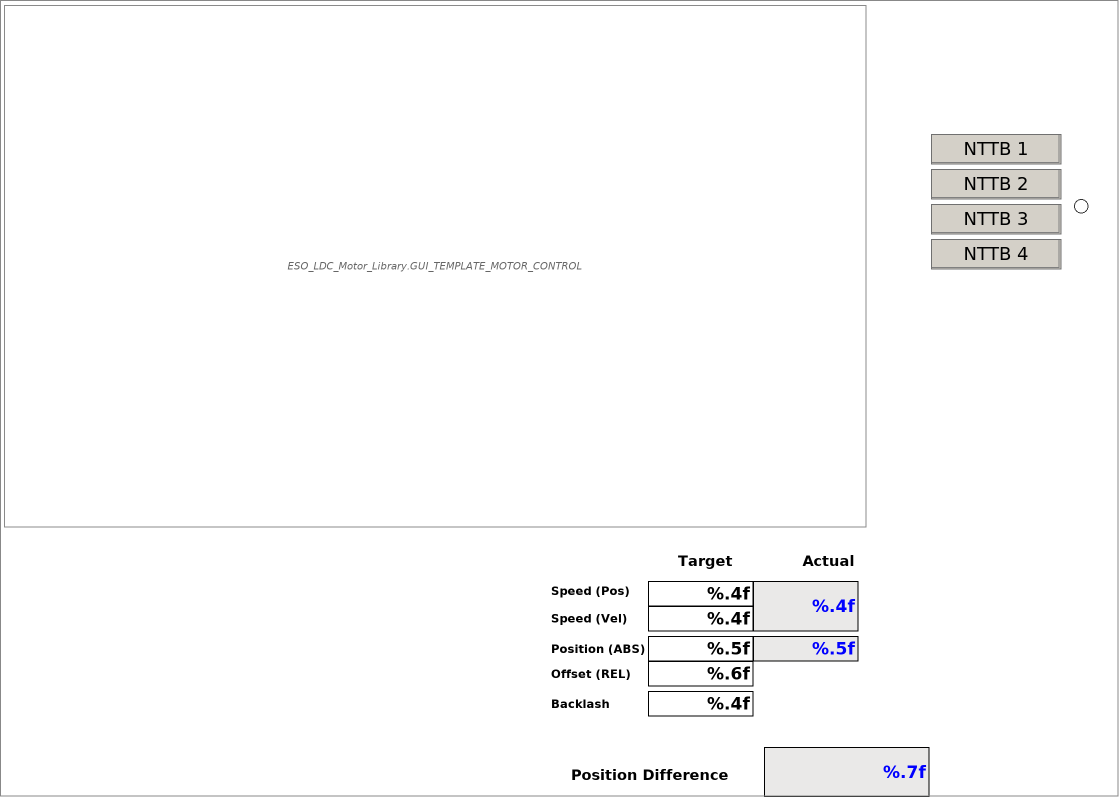
VISUALIZATION GUI_NOTT_TILT_B_CTRL  // 1119x797
    Frame (4,5 862x522)
        shows ESO_LDC_Motor_Library.GUI_TEMPLATE_MOTOR_CONTROL(m_Instance := MAIN.nott_ics.TipTilt.ptrTiltActuatorsB[MAIN.nott_ics.TipTilt.guiTiltActuatorsBIndex]^)
    Rectangle (548,581 95x20), "Speed (Pos)"
    Rectangle (753,636 105x25), "%.5f", text variable: MAIN.nott_ics.Delay_Lines.ptrDelayLines[MAIN.nott_ics.Delay_Lines.guiShutterIndex]^.stat.lrPosActual, input disabled if: false
    Rectangle (675,551 190x20), "Target Actual"
    Rectangle (548,639 95x20), "Position (ABS)"
    Rectangle (753,581 105x50), "%.4f", text variable: MAIN.nott_ics.Delay_Lines.ptrDelayLines[MAIN.nott_ics.Delay_Lines.guiShutterIndex]^.stat.lrVelActual, input disabled if: false
    Rectangle (648,606 105x25), "%.4f", text variable: MAIN.nott_ics.Delay_Lines.ptrDelayLines[MAIN.nott_ics.Delay_Lines.guiShutterIndex]^.ctrl.lrVelocity
        OnMouseDown: write the text variable via Default
    Rectangle (548,694 95x20), "Backlash"
    Rectangle (648,691 105x25), "%.4f", text variable: MAIN.nott_ics.Delay_Lines.ptrDelayLines[MAIN.nott_ics.Delay_Lines.guiShutterIndex]^.cfg.lrBacklash
        OnMouseDown: write the text variable via Default
    Rectangle (548,606 95x25), "Speed (Vel)"
    Rectangle (648,636 105x25), "%.5f", tooltip "Absolute position used by "MOVE ABS"", text variable: MAIN.nott_ics.Delay_Lines.ptrDelayLines[MAIN.nott_ics.Delay_Lines.guiShutterIndex]^.ctrl.lrPosition
        OnMouseDown: write the text variable via Default
    Rectangle (648,581 105x25), "%.4f", text variable: MAIN.nott_ics.Delay_Lines.ptrDelayLines[MAIN.nott_ics.Delay_Lines.guiShutterIndex]^.cfg.lrDefaultVelocity
        OnMouseDown: write the text variable via Default
    Rectangle (548,664 95x20), "Offset (REL)"
    Rectangle (648,661 105x25), "%.6f", tooltip "Relative offset used by "MOVE REL"", text variable: MAIN.nott_ics.Delay_Lines.ptrDelayLines[MAIN.nott_ics.Delay_Lines.guiShutterIndex]^.ctrl.lrOffset
        OnMouseDown: write the text variable via Default
    Rectangle (764,747 165x50), "%.7f", text variable: MAIN.nott_ics.Delay_Lines.ptrDelayLines[MAIN.nott_ics.Delay_Lines.guiShutterIndex]^.stat.lrPosError, input disabled if: false
    Rectangle (568,765 190x20), "Position Difference"
    RadioButton (1072,136 47x140), variable: MAIN.nott_ics.TipTilt.guiTiltActuatorsBIndex-1
        Areas[0]: Text=Radiobutton
        Areas[1]: Text=Radiobutton
    Button (931,134 130x30), "NTTB 1"
        OnMouseClick: execute { MAIN.nott_ics.TipTilt.guiTiltActuatorsBIndex := 1; }
    Button (931,169 130x30), "NTTB 2"
        OnMouseClick: execute { MAIN.nott_ics.TipTilt.guiTiltActuatorsBIndex := 2; }
    Button (931,204 130x30), "NTTB 3"
        OnMouseClick: execute { MAIN.nott_ics.TipTilt.guiTiltActuatorsBIndex := 3; }
    Button (931,239 130x30), "NTTB 4"
        OnMouseClick: execute { MAIN.nott_ics.TipTilt.guiTiltActuatorsBIndex := 4; }
END_VISUALIZATION

// ---- VISUs/Templates/MOTOR_CONTROL.TcVIS
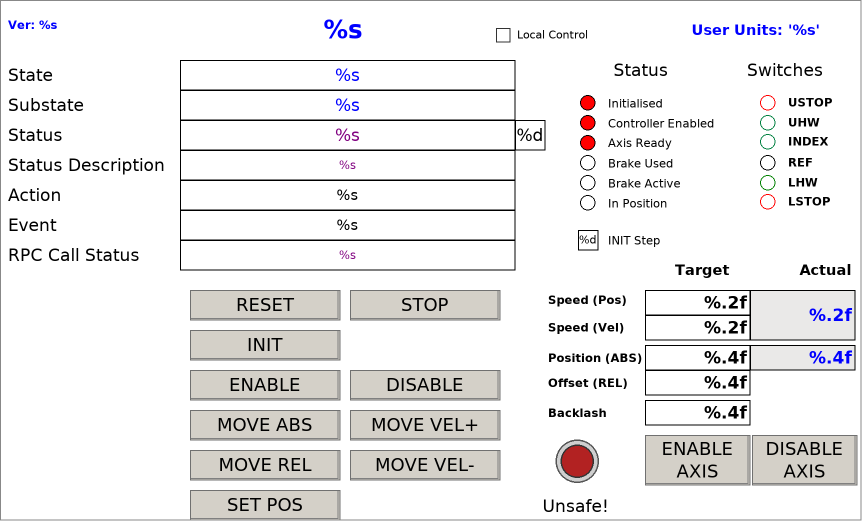
VISUALIZATION MOTOR_CONTROL  // 862x521
VAR_IN_OUT
	m_Instance:	FB_MOTOR;
END_VAR
    Rectangle (180,60 335x30), "%s", text variable: m_Instance.stat.sState
    Rectangle (180,90 335x30), "%s", text variable: m_Instance.stat.sSubstate
    Button (190,290 150x30), "RESET", input disabled if: NOT m_Instance.stat.bLocal OR NOT m_Instance.in_bSafe
        OnMouseDown: execute {
            m_Instance.ctrl.bLocalCmd := TRUE;
            m_Instance.ctrl.nCommand := E_MOTOR_COMMAND.RESET;
            m_Instance.ctrl.bExecute := TRUE;
        }
    Button (190,330 150x30), "INIT", input disabled if: NOT m_Instance.stat.bLocal OR NOT m_Instance.in_bSafe
        OnMouseDown: execute {
            m_Instance.ctrl.bLocalCmd := TRUE;
            m_Instance.ctrl.nCommand := E_MOTOR_COMMAND.INIT;
            m_Instance.ctrl.bExecute := TRUE;
        }
    Button (350,290 150x30), "STOP", input disabled if: NOT m_Instance.stat.bLocal OR NOT m_Instance.in_bSafe
        OnMouseDown: execute {
            m_Instance.ctrl.bLocalCmd := TRUE;
            m_Instance.ctrl.nCommand := E_MOTOR_COMMAND.STOP;
            m_Instance.ctrl.bExecute := TRUE;
        }
    Button (190,370 150x30), "ENABLE", input disabled if: NOT m_Instance.stat.bLocal OR NOT m_Instance.in_bSafe
        OnMouseDown: execute {
            m_Instance.ctrl.bLocalCmd := TRUE;
            m_Instance.ctrl.nCommand := E_MOTOR_COMMAND.ENABLE;
            m_Instance.ctrl.bExecute := TRUE;
        }
    Button (350,370 150x30), "DISABLE", input disabled if: NOT m_Instance.stat.bLocal OR NOT m_Instance.in_bSafe
        OnMouseDown: execute {
            m_Instance.ctrl.bLocalCmd := TRUE;
            m_Instance.ctrl.nCommand := E_MOTOR_COMMAND.DISABLE;
            m_Instance.ctrl.bExecute := TRUE;
        }
    Button (190,410 150x30), "MOVE ABS", input disabled if: NOT m_Instance.stat.bLocal OR NOT m_Instance.in_bSafe
        OnMouseDown: execute {
            m_Instance.ctrl.bLocalCmd := TRUE;
            m_Instance.ctrl.lrVelocity:=(m_Instance.cfg.lrDefaultVelocity);
            m_Instance.ctrl.nCommand := E_MOTOR_COMMAND.MOTOR_MOVE;
            m_Instance.ctrl.nMoveType := E_MOTOR_MOVE_TYPE.ABSOLUTE;
            m_Instance.ctrl.bExecute := TRUE;
        }
    Button (350,410 150x30), "MOVE VEL+", input disabled if: NOT m_Instance.stat.bLocal OR NOT m_Instance.in_bSafe
        OnMouseDown: execute {
            m_Instance.ctrl.bLocalCmd := TRUE;
            m_Instance.ctrl.nCommand := E_MOTOR_COMMAND.MOTOR_MOVE;
            m_Instance.ctrl.nMoveType := E_MOTOR_MOVE_TYPE.VELOCITY;
            m_Instance.ctrl.nDirection := MC_Positive_Direction;
            m_Instance.ctrl.bExecute := TRUE;
        }
    Rectangle (5,60 170x30), "State"
    Rectangle (5,90 170x30), "Substate"
    Rectangle (180,120 335x30), "%s", text variable: m_Instance.stat.sStatus
    Rectangle (180,150 335x30), "%s", tooltip "Additional information mostly used for description of errors", text variable: m_Instance.stat.sErrorText
    Rectangle (5,120 170x30), "Status"
    Rectangle (5,150 170x30), "Status Description"
    Rectangle (180,180 335x30), "%s", text variable: m_Instance.stat.sActionDesc
    Rectangle (180,210 335x30), "%s", text variable: m_Instance.stat.sEventDesc
    Rectangle (5,180 170x30), "Action"
    Rectangle (5,210 170x30), "Event"
    Rectangle (227,12 232x35), "%s", text variable: m_Instance.sName
    Checkbox (494,20 116x30), "Local Control", variable: m_Instance.stat.bLocal
    Rectangle (595,55 92x30), "Status"
    Rectangle (515,120 30x30), "%d", text variable: m_Instance.stat.nStatus
    Rectangle (739,55 92x30), "Switches"
    Button (350,450 150x30), "MOVE VEL-", input disabled if: NOT m_Instance.stat.bLocal OR NOT m_Instance.in_bSafe
        OnMouseDown: execute {
            m_Instance.ctrl.bLocalCmd := TRUE;
            m_Instance.ctrl.nCommand := E_MOTOR_COMMAND.MOTOR_MOVE;
            m_Instance.ctrl.nMoveType := E_MOTOR_MOVE_TYPE.VELOCITY;
            m_Instance.ctrl.nDirection := MC_Negative_Direction;
            m_Instance.ctrl.bExecute := TRUE;
        }
    Button (190,450 150x30), "MOVE REL", input disabled if: NOT m_Instance.stat.bLocal OR NOT m_Instance.in_bSafe
        OnMouseDown: execute {
            m_Instance.ctrl.bLocalCmd := TRUE;
            m_Instance.ctrl.lrVelocity:=(m_Instance.cfg.lrDefaultVelocity);
            m_Instance.ctrl.nCommand := E_MOTOR_COMMAND.MOTOR_MOVE;
            m_Instance.ctrl.nMoveType := E_MOTOR_MOVE_TYPE.RELATIVE;
            m_Instance.ctrl.bExecute := TRUE;
        }
    Button (190,490 150x30), "SET POS", input disabled if: NOT m_Instance.stat.bLocal OR NOT m_Instance.in_bSafe
        OnMouseDown: execute {
            m_Instance.ctrl.bLocalCmd := TRUE;
            m_Instance.ctrl.nCommand := E_MOTOR_COMMAND.SET_POSITION;
            m_Instance.ctrl.bExecute := TRUE;
        }
    Rectangle (785,95 50x15), "USTOP"
    Ellipse (760,95 15x15), colour toggle: m_Instance.stat.signals[5].bActive
    Ellipse (760,115 15x15), colour toggle: m_Instance.stat.signals[4].bActive
    Ellipse (760,175 15x15), colour toggle: m_Instance.stat.signals[1].bActive
    Ellipse (760,194 15x15), colour toggle: m_Instance.stat.signals[0].bActive
    Ellipse (760,155 15x15), colour toggle: m_Instance.stat.signals[2].bActive
    Rectangle (785,134 50x15), "INDEX"
    Rectangle (785,115 50x15), "UHW"
    Rectangle (785,155 50x15), "REF"
    Rectangle (785,175 50x15), "LHW"
    Rectangle (785,194 50x15), "LSTOP"
    Ellipse (760,134 15x15), colour toggle: m_Instance.stat.signals[3].bActive
    Rectangle (545,290 95x20), "Speed (Pos)"
    Rectangle (750,345 105x25), "%.4f", text variable: m_Instance.stat.lrPosActual, input disabled if: false
    Rectangle (672,260 190x20), "Target Actual"
    Rectangle (545,348 95x20), "Position (ABS)"
    Rectangle (750,290 105x50), "%.2f", text variable: m_Instance.stat.lrVelActual, input disabled if: false
    Rectangle (645,315 105x25), "%.2f", text variable: m_Instance.ctrl.lrVelocity
        OnMouseDown: write the text variable via Default
    Rectangle (545,403 95x20), "Backlash"
    Rectangle (645,400 105x25), "%.4f", text variable: m_Instance.cfg.lrBacklash
        OnMouseDown: write the text variable via Default
    Rectangle (545,315 95x25), "Speed (Vel)"
    Rectangle (645,345 105x25), "%.4f", tooltip "Absolute position used by "MOVE ABS"", text variable: m_Instance.ctrl.lrPosition
        OnMouseDown: write the text variable via Default
    Rectangle (645,290 105x25), "%.2f", text variable: m_Instance.cfg.lrDefaultVelocity
        OnMouseDown: write the text variable via Default
    Rectangle (605,171 90x25), "Brake Active"
    Ellipse (580,175 15x15), tooltip "RED = Applied BLANK = Released", colour toggle: (m_Instance.stat.bBrakeActive) <> 0
    Ellipse (580,95 15x15), tooltip "GREEN = Initialised RED = Not Initialised", text variable: m_Instance.stat.bInitialised, colour toggle: m_Instance.stat.bInitialised
    Rectangle (605,91 90x25), "Initialised"
    Rectangle (605,111 125x25), "Controller Enabled"
    Rectangle (605,131 90x24), "Axis Ready"
    Rectangle (605,151 90x25), "Brake Used"
    Ellipse (580,115 15x15), tooltip "GREEN = Enabled RED = Disabled", colour toggle: m_Instance.stat.bEnabled
    Ellipse (580,135 15x15), tooltip "GREEN = Ready RED = Not Ready", colour toggle: m_Instance.stat.bAxisReady
    Ellipse (580,155 15x15), tooltip "BLUE = Used BLANK = Not Used", colour toggle: m_Instance.cfg.bUseBrake
    Rectangle (578,230 20x20), "%d", text variable: m_Instance.stat.nInitStep
    Rectangle (605,228 90x25), "INIT Step"
    Rectangle (5,240 170x30), "RPC Call Status"
    Rectangle (180,240 335x30), "%s", text variable: m_Instance.stat.sRPCErrorText
    Rectangle (605,191 90x25), "In Position"
    Ellipse (580,195 15x15), tooltip "GREEN = In Position BLANK = Not In Position (or not used)", colour toggle: (m_Instance.stat.bInPosition) <> 0
    Button (645,435 105x50), "ENABLE AXIS", input disabled if: NOT m_Instance.stat.bLocal OR NOT m_Instance.in_bSafe
        OnMouseDown: execute { m_Instance.stat.bEnabled := TRUE; }
    Button (752,435 105x50), "DISABLE AXIS", input disabled if: NOT m_Instance.stat.bLocal OR NOT m_Instance.in_bSafe
        OnMouseDown: execute { m_Instance.stat.bEnabled := FALSE; }
    Rectangle (620,15 203x30), "User Units: '%s'", text variable: m_Instance.stat.axis.sUnits
    Rectangle (5,10 99x30), "Ver: %s", tooltip "'Motor.library version'", text variable: m_Instance.stat.sLibVersion, input disabled if: true
    Rectangle (545,373 95x20), "Offset (REL)"
    Rectangle (645,370 105x25), "%.4f", tooltip "Relative offset used by "MOVE REL"", text variable: m_Instance.ctrl.lrOffset
        OnMouseDown: write the text variable via Default
    Lamp1 (552,436 50x50), tooltip "If active, it is not safe to operate the motor.", variable: NOT m_Instance.in_bSafe, invisible if: m_Instance.in_bSafe, style: Lamp-Lamp1-Red
    Rectangle (526,491 100x30), "Unsafe!", invisible if: m_Instance.in_bSafe
END_VISUALIZATION
